// TIA Portal V19 export
DATA_BLOCK "PostPunchingMatCounter_PERS"   // DB147
{ DB_Accessible_From_OPC_UA := 'FALSE' }
// stored: DBAccessibleFromOPCUA false, MemoryReserve 100
   VAR RETAIN
      PersistentValues : "MatCountPersistent";
   END_VAR
BEGIN
   PersistentValues.Data.AxPosition := 0.0;
   PersistentValues.Data.AxPositionPrevious := 230131.927;
   PersistentValues.Data.FAK := 1.00085820598793;
   PersistentValues.Data.CounterValueInit := 233955.205122556;
   PersistentValues.Data.CounterOffset := 3625.77752479035;
   PersistentValues.Data.CounterValue := 233955.205122556;
   PersistentValues.Data.FAKPrevious := 1.00074560970077;
   PersistentValues.Data.AX_MODULE := 1000000.0;
   PersistentValues.Data.COUNTER_MODULE := 1000000.0;
   PersistentValues.Par.FAK := 1.00085820598793;
END_DATA_BLOCK
